DATA_BLOCK "DB2045_TQ_AE"
TITLE = DB2045_TQ_AE
{ S7_Optimized_Access := 'FALSE' }
AUTHOR : HCR
FAMILY : ZeusControl
VERSION : 1.0
   STRUCT
      AE { S7_SetPoint := 'False'} : Array[0.."N_MAX_DISP_TQ_AE"] of "UDT_ZC_DISP_TQ_AE";
      Mux { S7_SetPoint := 'False'} : Array[0.."N_MAX_MUX_DISP"] of "UDT_ZC_DISP_MUX_TQ_AE";
      Agrup : Array[0.."N_MAX_DISP_AGRUP"] of "UDT_ZC_DISP_AGRUP";
   END_STRUCT;


BEGIN
   AE[0].Estado_AutoMan := FALSE;
   AE[0].Orden_Manual := FALSE;
   AE[0].Orden_CIP := FALSE;
   AE[0].Orden_Produccion := FALSE;
   AE[0].Orden_Vaciado := FALSE;
   AE[0].Alarma_PresionAlta := FALSE;
   AE[0].Alarma_PresionBaja := FALSE;
   AE[0].Alarma_Configuracion := FALSE;
   AE[0].Salida_ValvulaVenteo := FALSE;
   AE[0].Salida_ValvulaEsteril := FALSE;
   AE[0].Salida_ValvulaDucha := FALSE;
   AE[0].Aux_DuchaFlipActivo := FALSE;
   AE[0].Aux_DuchaFlopActivo := TRUE;
   AE[0].Aux_DuchaFlanco := FALSE;
   AE[0].Aux_DuchaSalidaFlip := FALSE;
   AE[0].Aux_DuchaSalidaFlop := FALSE;
   AE[0].Config_Habilitar := FALSE;
   AE[0].Config_HabilitarAlarmas := FALSE;
   AE[0].Aux_oldOrdenManual := FALSE;
   AE[0].Aux_oldAutoMan := FALSE;
   AE[0].Config_GrupoAlarma := 0;
   AE[0].Estado_ValorPresion := 0.0;
   AE[0].Config_PresionMaxTrabajo := 0.0;
   AE[0].Config_PresionMinTrabajo := 0.0;
   AE[0].Config_PresionMaxAlarma := 0.0;
   AE[0].Config_PresionMinAlarma := 0.0;
   AE[0].Tiempos_SetPointAlarmaMaxPresion := 0;
   AE[0].Tiempos_SetPointAlarmaMinPresion := 0;
   AE[0].Tiempos_AlarmaMaxPresion := 0;
   AE[0].Tiempos_AlarmaMinPresion := 0;
   AE[0].Tiempos_SetPointFlipDucha := 0;
   AE[0].Tiempos_SetPointFlopDucha := 0;
   AE[0].Tiempos_DuchaTiempoFlip := 0;
   AE[0].Tiempos_DuchaTiempoFlop := 0;
   AE[1].Estado_AutoMan := TRUE;
   AE[1].Orden_Manual := FALSE;
   AE[1].Orden_CIP := FALSE;
   AE[1].Orden_Produccion := FALSE;
   AE[1].Orden_Vaciado := FALSE;
   AE[1].Alarma_PresionAlta := FALSE;
   AE[1].Alarma_PresionBaja := FALSE;
   AE[1].Alarma_Configuracion := FALSE;
   AE[1].Salida_ValvulaVenteo := FALSE;
   AE[1].Salida_ValvulaEsteril := FALSE;
   AE[1].Salida_ValvulaDucha := FALSE;
   AE[1].Aux_DuchaFlipActivo := FALSE;
   AE[1].Aux_DuchaFlopActivo := TRUE;
   AE[1].Aux_DuchaFlanco := FALSE;
   AE[1].Aux_DuchaSalidaFlip := FALSE;
   AE[1].Aux_DuchaSalidaFlop := FALSE;
   AE[1].Config_Habilitar := TRUE;
   AE[1].Config_HabilitarAlarmas := TRUE;
   AE[1].Aux_oldOrdenManual := FALSE;
   AE[1].Aux_oldAutoMan := TRUE;
   AE[1].Config_GrupoAlarma := 0;
   AE[1].Estado_ValorPresion := 0.0003616898;
   AE[1].Config_PresionMaxTrabajo := 0.2;
   AE[1].Config_PresionMinTrabajo := 0.1;
   AE[1].Config_PresionMaxAlarma := 0.6;
   AE[1].Config_PresionMinAlarma := 0.05;
   AE[1].Tiempos_SetPointAlarmaMaxPresion := 10;
   AE[1].Tiempos_SetPointAlarmaMinPresion := 60;
   AE[1].Tiempos_AlarmaMaxPresion := 0;
   AE[1].Tiempos_AlarmaMinPresion := 649;
   AE[1].Tiempos_SetPointFlipDucha := 0;
   AE[1].Tiempos_SetPointFlopDucha := 0;
   AE[1].Tiempos_DuchaTiempoFlip := 0;
   AE[1].Tiempos_DuchaTiempoFlop := 0;
   Mux[0].Habilitar := TRUE;
   Mux[0].ExisteCambio := FALSE;
   Mux[0].MaxVisible := FALSE;
   Mux[0].Index := 0;
   Mux[0].oldIndex := 0;
   Mux[0].AE.Estado_AutoMan := FALSE;
   Mux[0].AE.Orden_Manual := FALSE;
   Mux[0].AE.Orden_CIP := FALSE;
   Mux[0].AE.Orden_Produccion := FALSE;
   Mux[0].AE.Orden_Vaciado := FALSE;
   Mux[0].AE.Alarma_PresionAlta := FALSE;
   Mux[0].AE.Alarma_PresionBaja := FALSE;
   Mux[0].AE.Alarma_Configuracion := FALSE;
   Mux[0].AE.Salida_ValvulaVenteo := FALSE;
   Mux[0].AE.Salida_ValvulaEsteril := FALSE;
   Mux[0].AE.Salida_ValvulaDucha := FALSE;
   Mux[0].AE.Aux_DuchaFlipActivo := FALSE;
   Mux[0].AE.Aux_DuchaFlopActivo := TRUE;
   Mux[0].AE.Aux_DuchaFlanco := FALSE;
   Mux[0].AE.Aux_DuchaSalidaFlip := FALSE;
   Mux[0].AE.Aux_DuchaSalidaFlop := FALSE;
   Mux[0].AE.Config_Habilitar := FALSE;
   Mux[0].AE.Config_HabilitarAlarmas := FALSE;
   Mux[0].AE.Aux_oldOrdenManual := FALSE;
   Mux[0].AE.Aux_oldAutoMan := FALSE;
   Mux[0].AE.Config_GrupoAlarma := 0;
   Mux[0].AE.Estado_ValorPresion := 0.0;
   Mux[0].AE.Config_PresionMaxTrabajo := 0.0;
   Mux[0].AE.Config_PresionMinTrabajo := 0.0;
   Mux[0].AE.Config_PresionMaxAlarma := 0.0;
   Mux[0].AE.Config_PresionMinAlarma := 0.0;
   Mux[0].AE.Tiempos_SetPointAlarmaMaxPresion := 0;
   Mux[0].AE.Tiempos_SetPointAlarmaMinPresion := 0;
   Mux[0].AE.Tiempos_AlarmaMaxPresion := 0;
   Mux[0].AE.Tiempos_AlarmaMinPresion := 0;
   Mux[0].AE.Tiempos_SetPointFlipDucha := 0;
   Mux[0].AE.Tiempos_SetPointFlopDucha := 0;
   Mux[0].AE.Tiempos_DuchaTiempoFlip := 0;
   Mux[0].AE.Tiempos_DuchaTiempoFlop := 0;
   Mux[1].Habilitar := TRUE;
   Mux[1].ExisteCambio := FALSE;
   Mux[1].MaxVisible := FALSE;
   Mux[1].Index := 0;
   Mux[1].oldIndex := 0;
   Mux[1].AE.Estado_AutoMan := FALSE;
   Mux[1].AE.Orden_Manual := FALSE;
   Mux[1].AE.Orden_CIP := FALSE;
   Mux[1].AE.Orden_Produccion := FALSE;
   Mux[1].AE.Orden_Vaciado := FALSE;
   Mux[1].AE.Alarma_PresionAlta := FALSE;
   Mux[1].AE.Alarma_PresionBaja := FALSE;
   Mux[1].AE.Alarma_Configuracion := FALSE;
   Mux[1].AE.Salida_ValvulaVenteo := FALSE;
   Mux[1].AE.Salida_ValvulaEsteril := FALSE;
   Mux[1].AE.Salida_ValvulaDucha := FALSE;
   Mux[1].AE.Aux_DuchaFlipActivo := FALSE;
   Mux[1].AE.Aux_DuchaFlopActivo := TRUE;
   Mux[1].AE.Aux_DuchaFlanco := FALSE;
   Mux[1].AE.Aux_DuchaSalidaFlip := FALSE;
   Mux[1].AE.Aux_DuchaSalidaFlop := FALSE;
   Mux[1].AE.Config_Habilitar := FALSE;
   Mux[1].AE.Config_HabilitarAlarmas := FALSE;
   Mux[1].AE.Aux_oldOrdenManual := FALSE;
   Mux[1].AE.Aux_oldAutoMan := FALSE;
   Mux[1].AE.Config_GrupoAlarma := 0;
   Mux[1].AE.Estado_ValorPresion := 0.0;
   Mux[1].AE.Config_PresionMaxTrabajo := 0.0;
   Mux[1].AE.Config_PresionMinTrabajo := 0.0;
   Mux[1].AE.Config_PresionMaxAlarma := 0.0;
   Mux[1].AE.Config_PresionMinAlarma := 0.0;
   Mux[1].AE.Tiempos_SetPointAlarmaMaxPresion := 0;
   Mux[1].AE.Tiempos_SetPointAlarmaMinPresion := 0;
   Mux[1].AE.Tiempos_AlarmaMaxPresion := 0;
   Mux[1].AE.Tiempos_AlarmaMinPresion := 0;
   Mux[1].AE.Tiempos_SetPointFlipDucha := 0;
   Mux[1].AE.Tiempos_SetPointFlopDucha := 0;
   Mux[1].AE.Tiempos_DuchaTiempoFlip := 0;
   Mux[1].AE.Tiempos_DuchaTiempoFlop := 0;
   Agrup[0].AlgunaEnManual := TRUE;
   Agrup[0].AlgunaAlarma := FALSE;
   Agrup[0].NuevaAlarma := FALSE;
   Agrup[1].AlgunaEnManual := FALSE;
   Agrup[1].AlgunaAlarma := FALSE;
   Agrup[1].NuevaAlarma := FALSE;

END_DATA_BLOCK

